{attribute 'TcGenerated'}
// This function has been automatically generated from the project information.
VAR_GLOBAL CONSTANT
    {attribute 'const_non_replaced'}
    {attribute 'linkalways'}
    stLibVersion_lcls_twincat_optics : ST_LibVersion := (iMajor := 0, iMinor := 4, iBuild := 1, iRevision := 0, sVersion := '0.4.1');
END_VAR

(* stored: Version 1.1.0.1, ProductVersion 3.1.4022.18
   GVL Global_Version: Id 955b45c6-8733-4e36-98ae-c5d0d98857db *)
